{attribute 'GeneratedUsingTerminal: EL5021-0000-0016'}
{attribute addProperty BoxType "EL5021-0000-0016"}
{attribute addProperty Id "ENC_StatusAT %I*ENC_Status_1E2673DC16ENC_ControlAT %Q*ENC_Control_64DD586E6WcStateAT %I*WcState_9091E0EB2InfoDataAT %I*InfoData_32EB74EA10"}
{attribute addProperty CRC "600991009"}
{attribute addProperty Size "34"}
TYPE EL5021_23D26521 EXTENDS EtcSlaveTerminalBase_947E5A46 :
STRUCT
	{attribute addProperty Name "ENC_Status"}
	ENC_Status : ENC_Status_1E2673DC;
	{attribute addProperty Name "ENC_Control"}
	ENC_Control : ENC_Control_64DD586E;
	{attribute addProperty Name "WcState"}
	WcState : WcState_9091E0EB;
	{attribute addProperty Name "InfoData"}
	InfoData : InfoData_32EB74EA;
END_STRUCT
END_TYPE

(* stored: Version 1.2.0.0, ProductVersion 3.1.4024.9
   DUT EL5021_23D26521: Id {fbc9c791-004c-49b6-afc9-fa02fda24fd3} *)
